Staubli VAL3: dioItem.pjx

--- dioItem.pjx ---
Parameters version=s7.2.1 stackSize=5000 millimeterUnit=true
Data file=dioItem.dtx

--- dioItem.dtx ---
public bool bActive
public string sID
public string sName
public dio dDio
public bool bEnable
